TYPE ST_Parameters :
STRUCT
END_STRUCT
END_TYPE

(* stored: Version 1.1.0.1, ProductVersion 3.1.4024.12
   DUT ST_Parameters: Id {b3925ad8-56dd-4650-bfc7-7fcbfe7184dd} *)
